// TIA Portal V17 export
// export: Created 2024-09-02T12:50:05.4870393Z, ExportSetting WithDefaults, DisplayName Totally Integrated Automation Portal, DisplayVersion V17, DisplayName TIA Portal Openness, DisplayVersion V17, DisplayName TIA Portal Version Control Interface, DisplayVersion V17, DisplayName STEP 7 Professional, DisplayVersion V17, DisplayName STEP 7 Safety, DisplayVersion V17, DisplayName WinCC Professional, DisplayVersion V17
FUNCTION_BLOCK "GraFB_Hand_01_10"   // FB1170, GRAPH
TITLE = GRAPH FB
AUTHOR : VAF
FAMILY : SK
NAME : SK
VERSION : 0.1
// Hand functions / Handfunktionen
// stored: AcknowledgeErrorsRequired true, AutoNumber true, ExtensionBlockName LTLL_ManualGraphExt, GraphVersion 4.0, InitialValuesAcquisition false, IsIECCheckEnabled false, LanguageInNetworks LAD, LockOperatingMode false, PermanentILProcessingInMANMode true, SetENOAutomatically false, SkipSteps false, UDAEnableTagReadback false, WithAlarmHandling true
   // inherited from GRAPH_BASE
   VAR
      OFF_SQ_BASE : Bool;
   END_VAR
   VAR_INPUT
      OFF_SQ : Bool;
      INIT_SQ : Bool;
      ACK_EF : Bool;
      S_PREV : Bool;
      S_NEXT : Bool;
      SW_AUTO : Bool;
      SW_TAP : Bool;
      SW_MAN : Bool;
      S_SEL : Int;
      S_ON : Bool;
      S_OFF : Bool;
      T_PUSH : Bool;
   END_VAR
   VAR_OUTPUT
      S_NO : Int;
      S_MORE : Bool;
      S_ACTIVE : Bool;
      ERR_FLT : Bool;
      AUTO_ON : Bool;
      TAP_ON : Bool;
      MAN_ON : Bool;
   END_VAR
   VAR
      extBlock { S7_SetPoint := 'True'} : "LTLL_ManualGraphExt";
   END_VAR
   VAR_TEMP
      t_FrgHand : Bool;   // Freigabe Handbetrieb / Enable manual operation
      t_Service : Bool;   // Servicebetrieb aktiv / Service operation active
   END_VAR
BEGIN
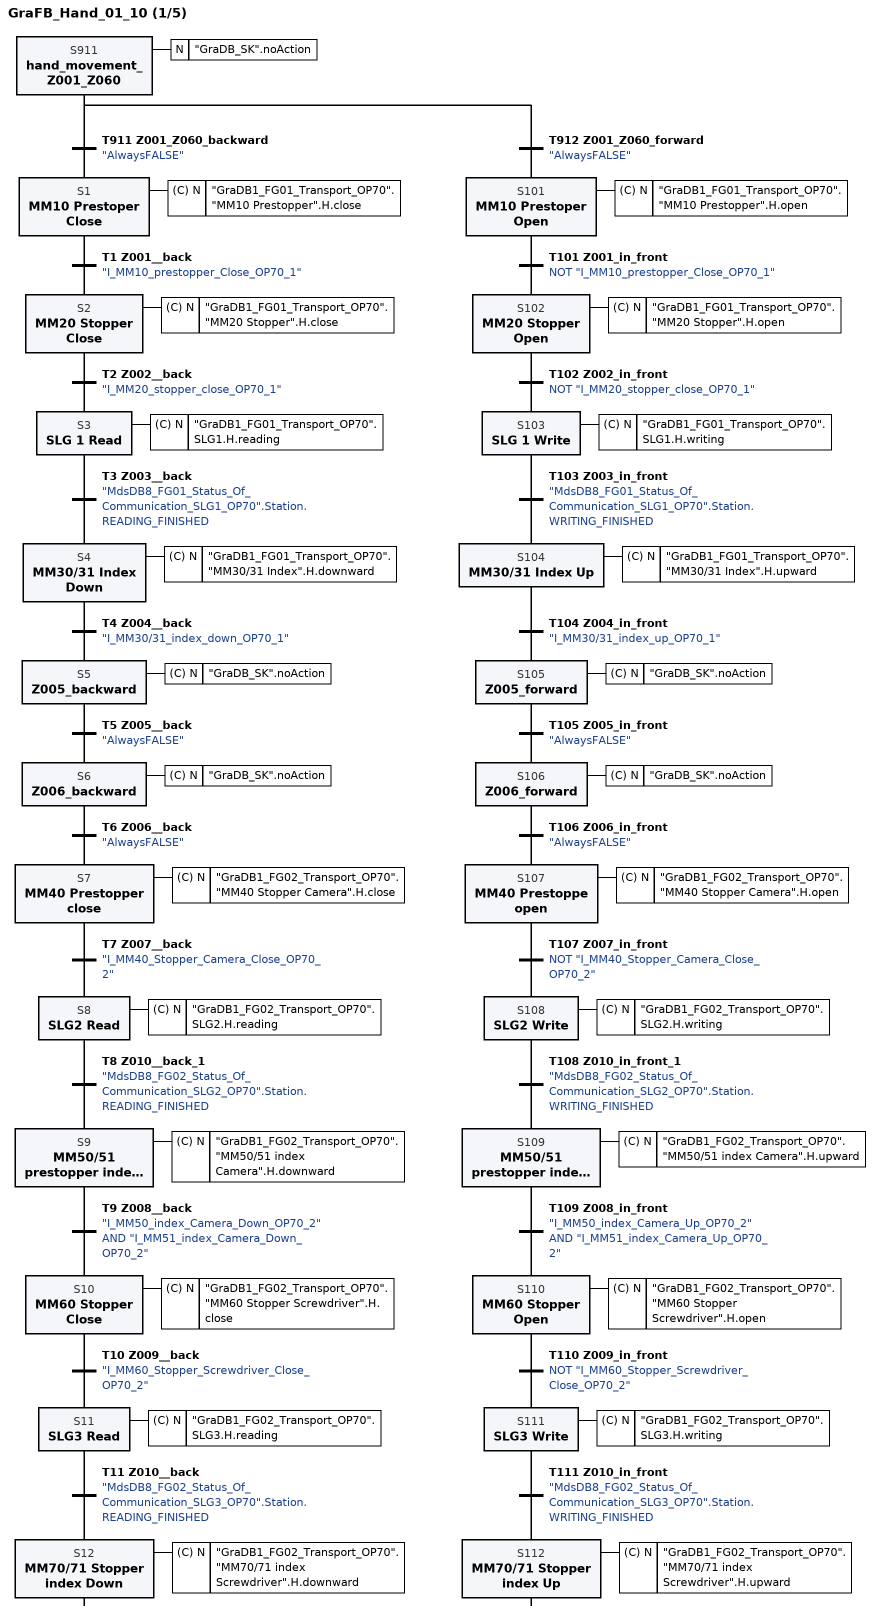
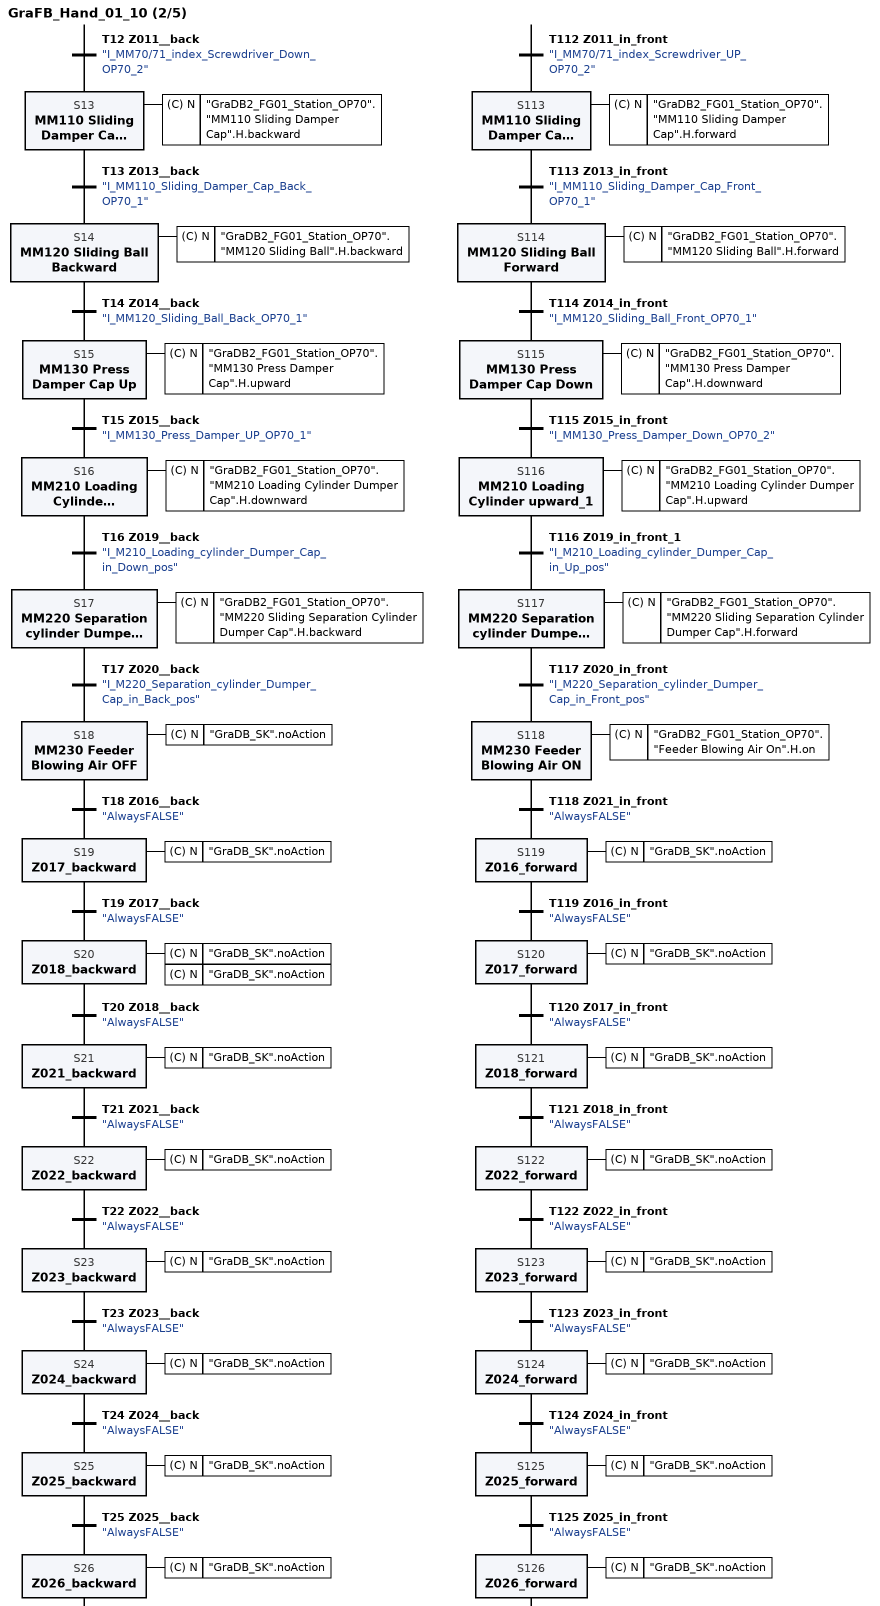
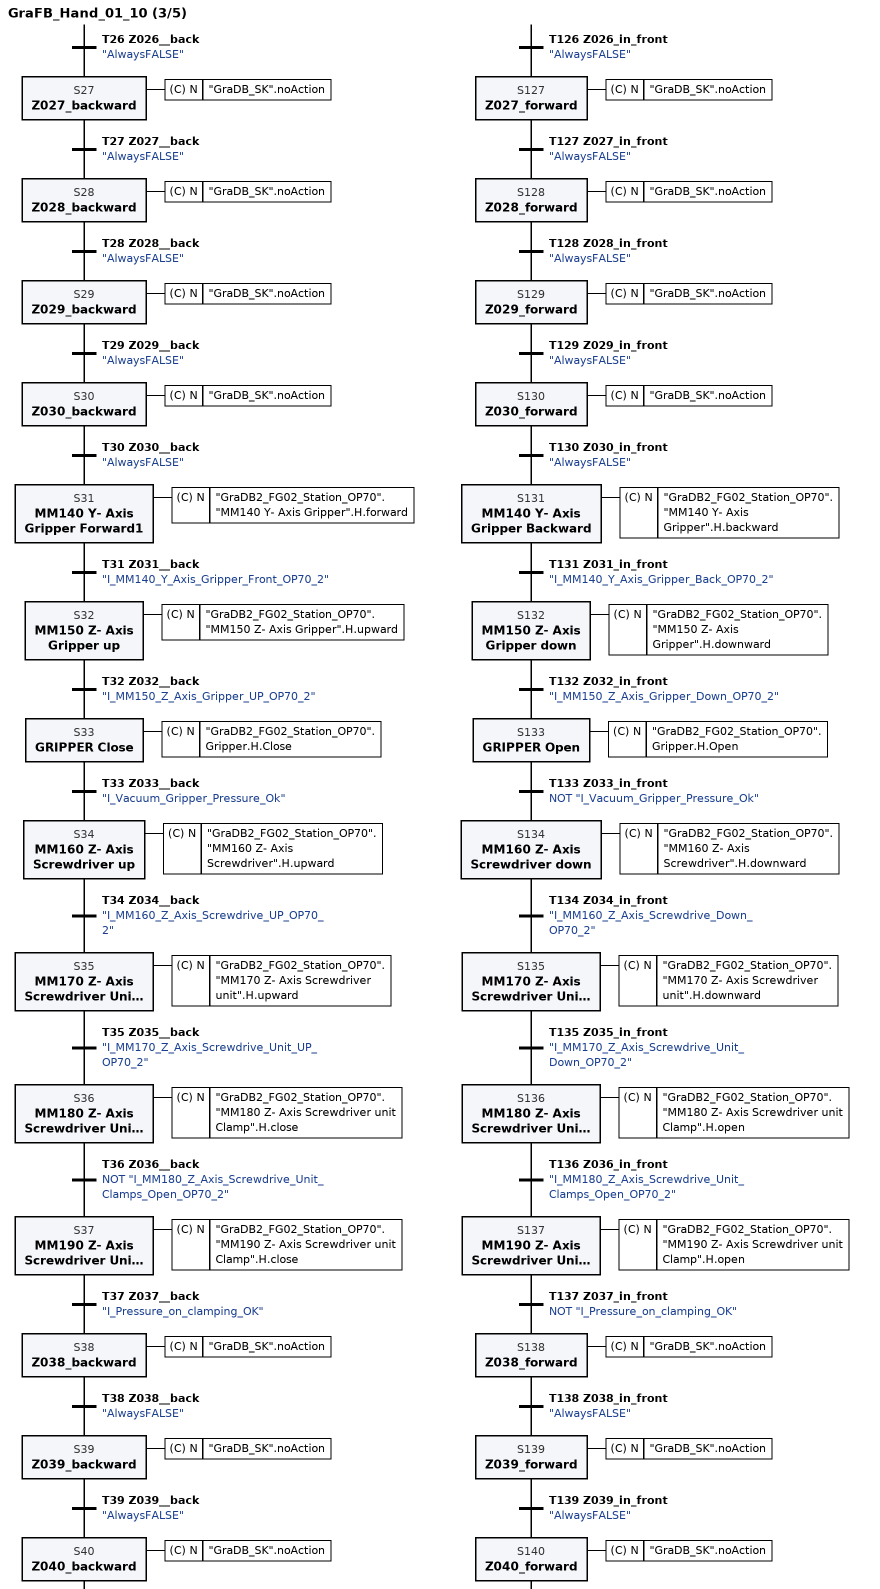
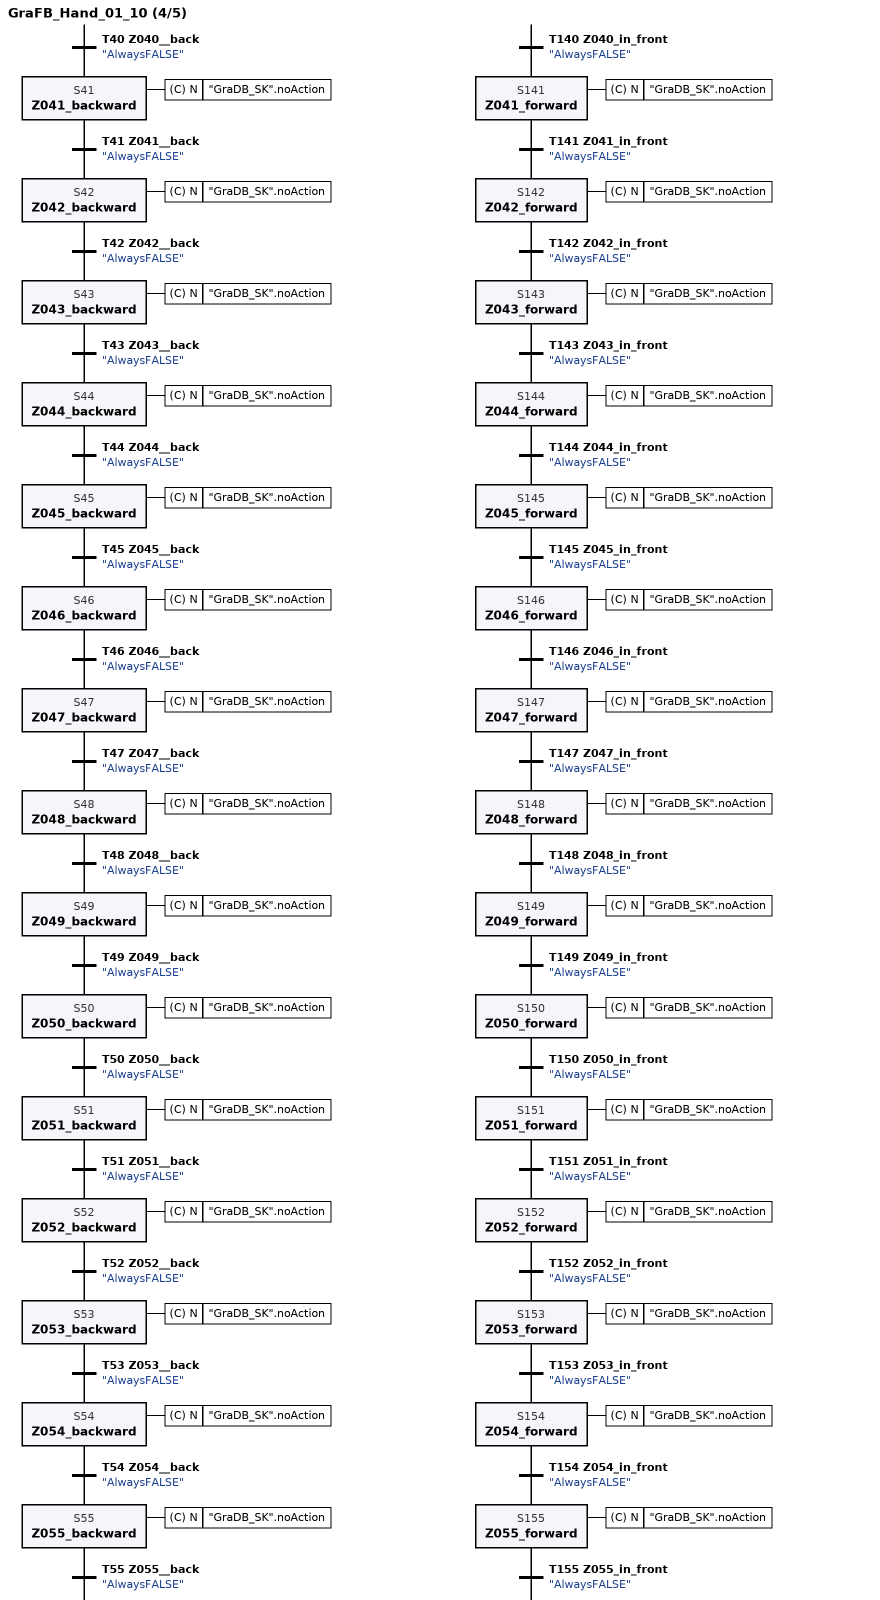
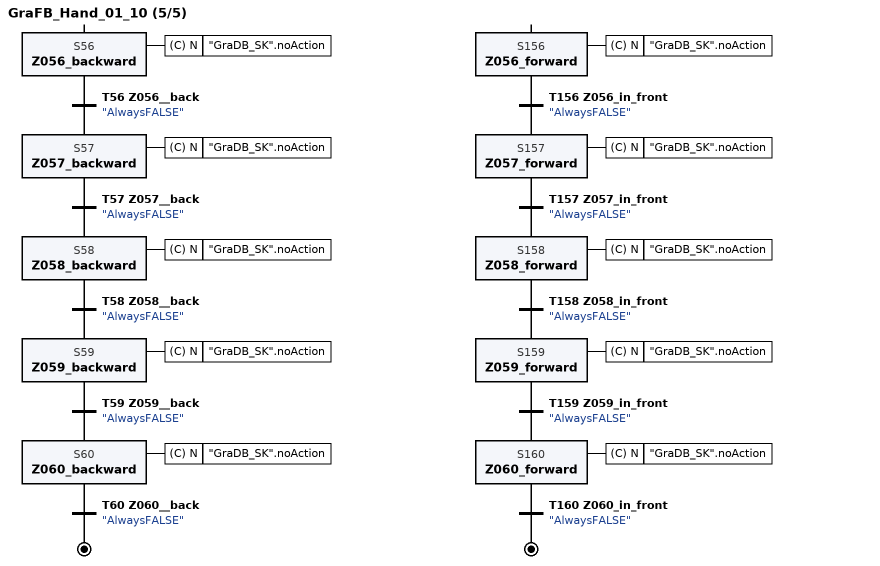
   // permanent pre-instructions
   NETWORK 1
   TITLE = HMI Lite Pass on data / HMI Lite Daten weiterreichen
      #extBlock.input := "LTLL_ManualGraphControl_OP70".screen[0].input;
   NETWORK 2
   TITLE = Instance DB Name query and pass on / Instanz DB Name abfragen und weiterreichen
      GetInstanceName(size := 0, OUT => #extBlock.input.instanceName);
   NETWORK 3
   TITLE = Interlocks Permanent machining, manual Approve and service / Interlocks Permanent Bearbeiten, Handfreigabe und Service
      IF NOT #RT_DATA.MOP.IL_PERM THEN #RT_DATA.MOP.IL_PERM := TRUE; END_IF;
      #t_FrgHand := "AnwDB_OperatingModes_OP70".BA[0]."mode_hand+start" AND "AnwDB_EKS_Data_OP70".EKS1.LEVEL_5_BK;
      #t_Service := "AnwDB_OperatingModes_OP70".BA[0].mode_service;

   // sequencer 1: Sequencer 1
   STEP hand_movement_Z001_Z060:   // S911, max time T#10S, warning time T#7S: Step commentary / Schrittkommentar
      interlock C := (none);   // hand_bereich_Z001_Z005
      supervision V := (none);   // hand_bereich_Z001_Z005
              N    "GraDB_SK".noAction
   END_STEP
   TRANSITION Z001_Z060_backward FROM hand_movement_Z001_Z060 TO "MM10 Prestoper Close"   // T911
      := "AlwaysFALSE";
   END_TRANSITION
   TRANSITION Z001_Z060_forward FROM hand_movement_Z001_Z060 TO "MM10 Prestoper Open"   // T912
      := "AlwaysFALSE";
   END_TRANSITION
   STEP "MM10 Prestoper Close":   // S1, max time T#10S, warning time T#7S
      interlock C := #t_FrgHand AND ("AlwaysTRUE" OR #t_Service);   // Z001_zur
      supervision V := NOT #Z001__back.TT AND (#"MM10 Prestoper Close".T > T#10S);   // Z001_zur
      (C)     N    "GraDB1_FG01_Transport_OP70"."MM10 Prestopper".H.close
   END_STEP
   TRANSITION Z001__back FROM "MM10 Prestoper Close" TO "MM20 Stopper Close"   // T1
      := "I_MM10_prestopper_Close_OP70_1";
   END_TRANSITION
   STEP "MM20 Stopper Close":   // S2, max time T#10S, warning time T#7S
      interlock C := #t_FrgHand AND ("AlwaysTRUE" OR #t_Service);   // Z002_zur
      supervision V := NOT #Z002__back.TT AND (#"MM20 Stopper Close".T > T#10S);   // Z002_zur
      (C)     N    "GraDB1_FG01_Transport_OP70"."MM20 Stopper".H.close
   END_STEP
   TRANSITION Z002__back FROM "MM20 Stopper Close" TO "SLG 1 Read"   // T2
      := "I_MM20_stopper_close_OP70_1";
   END_TRANSITION
   STEP "SLG 1 Read":   // S3, max time T#10S, warning time T#7S
      interlock C := #t_FrgHand AND "MdsDB8_FG01_Status_Of_Communication_SLG1_OP70".ASM.MDS_PRESENT;   // Z003_zur
      supervision V := NOT #Z003__back.TT AND (#"SLG 1 Read".T > T#10S);   // Z003_zur
      (C)     N    "GraDB1_FG01_Transport_OP70".SLG1.H.reading
   END_STEP
   TRANSITION Z003__back FROM "SLG 1 Read" TO "MM30/31 Index Down"   // T3
      := "MdsDB8_FG01_Status_Of_Communication_SLG1_OP70".Station.READING_FINISHED;
   END_TRANSITION
   STEP "MM30/31 Index Down":   // S4, max time T#10S, warning time T#7S
      interlock C := #t_FrgHand AND ("I_MM130_Press_Damper_UP_OP70_1" OR #t_Service);   // Z004_zur
      supervision V := NOT #Z004__back.TT AND (#"MM30/31 Index Down".T > T#10S);   // Z004_zur
      (C)     N    "GraDB1_FG01_Transport_OP70"."MM30/31 Index".H.downward
   END_STEP
   TRANSITION Z004__back FROM "MM30/31 Index Down" TO Z005_backward   // T4
      := "I_MM30/31_index_down_OP70_1";
   END_TRANSITION
   STEP Z005_backward:   // S5, max time T#10S, warning time T#7S
      interlock C := #t_FrgHand AND ("AlwaysFALSE" OR #t_Service);   // Z005_zur
      supervision V := NOT #Z005__back.TT AND (#Z005_backward.T > T#10S);   // Z005_zur
      (C)     N    "GraDB_SK".noAction
   END_STEP
   TRANSITION Z005__back FROM Z005_backward TO Z006_backward   // T5
      := "AlwaysFALSE";
   END_TRANSITION
   STEP "MM10 Prestoper Open":   // S101, max time T#10S, warning time T#7S
      interlock C := #t_FrgHand AND ((NOT "I_MM20_pallet_at_stopper_OP70_1" AND NOT "MdsDB8_FG01_Status_Of_Communication_SLG1_OP70".ASM.MDS_PRESENT AND "I_MM30/31_index_down_OP70_1" AND "I_MM130_Press_Damper_UP_OP70_1") OR NOT "I_MM10_pallet_at_prestopper_OP70_1" OR #t_Service);   // Z001_vor
      supervision V := NOT #Z001_in_front.TT AND (#"MM10 Prestoper Open".T > T#10S);   // Z001_vor
      (C)     N    "GraDB1_FG01_Transport_OP70"."MM10 Prestopper".H.open
   END_STEP
   TRANSITION Z001_in_front FROM "MM10 Prestoper Open" TO "MM20 Stopper Open"   // T101
      := NOT "I_MM10_prestopper_Close_OP70_1";
   END_TRANSITION
   STEP "MM20 Stopper Open":   // S102, max time T#10S, warning time T#7S
      interlock C := #t_FrgHand AND (("I_MM30/31_index_down_OP70_1" AND "I_MM130_Press_Damper_UP_OP70_1" AND NOT "I_MM40_pallet_at_Stopper_Camera_OP70_2" AND NOT "MdsDB8_FG02_Status_Of_Communication_SLG2_OP70".ASM.MDS_PRESENT AND "I_MM50_index_Camera_Down_OP70_2" AND "I_MM51_index_Camera_Down_OP70_2") OR (NOT "I_MM20_pallet_at_stopper_OP70_1" AND NOT "MdsDB8_FG01_Status_Of_Communication_SLG1_OP70".ASM.MDS_PRESENT) OR #t_Service);   // Z002_vor
      supervision V := NOT #Z002_in_front.TT AND (#"MM20 Stopper Open".T > T#10S);   // Z002_vor
      (C)     N    "GraDB1_FG01_Transport_OP70"."MM20 Stopper".H.open
   END_STEP
   TRANSITION Z002_in_front FROM "MM20 Stopper Open" TO "SLG 1 Write"   // T102
      := NOT "I_MM20_stopper_close_OP70_1";
   END_TRANSITION
   STEP "SLG 1 Write":   // S103, max time T#10S, warning time T#7S
      interlock C := #t_FrgHand AND "MdsDB8_FG01_Status_Of_Communication_SLG1_OP70".ASM.MDS_PRESENT AND "MdsDB8_FG01_Status_Of_Communication_SLG1_OP70".Station.READING_FINISHED;   // Z003_vor
      supervision V := NOT #Z003_in_front.TT AND (#"SLG 1 Write".T > T#10S);   // Z003_vor
      (C)     N    "GraDB1_FG01_Transport_OP70".SLG1.H.writing
   END_STEP
   TRANSITION Z003_in_front FROM "SLG 1 Write" TO "MM30/31 Index Up"   // T103
      := "MdsDB8_FG01_Status_Of_Communication_SLG1_OP70".Station.WRITING_FINISHED;
   END_TRANSITION
   STEP "MM30/31 Index Up":   // S104, max time T#10S, warning time T#7S
      interlock C := #t_FrgHand AND ("I_MM130_Press_Damper_UP_OP70_1" OR #t_Service);   // Z004_vor
      supervision V := NOT #Z004_in_front.TT AND (#"MM30/31 Index Up".T > T#10S);   // Z004_vor
      (C)     N    "GraDB1_FG01_Transport_OP70"."MM30/31 Index".H.upward
   END_STEP
   TRANSITION Z004_in_front FROM "MM30/31 Index Up" TO Z005_forward   // T104
      := "I_MM30/31_index_up_OP70_1";
   END_TRANSITION
   STEP Z005_forward:   // S105, max time T#10S, warning time T#7S
      interlock C := #t_FrgHand AND ("AlwaysFALSE" OR #t_Service);   // Z005_vor
      supervision V := NOT #Z005_in_front.TT AND (#Z005_forward.T > T#10S);   // Z005_vor
      (C)     N    "GraDB_SK".noAction
   END_STEP
   TRANSITION Z005_in_front FROM Z005_forward TO Z006_forward   // T105
      := "AlwaysFALSE";
   END_TRANSITION
   STEP Z006_backward:   // S6, max time T#10S, warning time T#7S: Cross transport 2 / Quertransport 2
      interlock C := #t_FrgHand AND ("AlwaysFALSE" OR #t_Service);   // Z006_zur
      supervision V := NOT #Z006__back.TT AND (#Z006_backward.T > T#10S);   // Z006_zur
      (C)     N    "GraDB_SK".noAction
   END_STEP
   TRANSITION Z006__back FROM Z006_backward TO "MM40 Prestopper close"   // T6
      := "AlwaysFALSE";
   END_TRANSITION
   STEP "MM40 Prestopper close":   // S7, max time T#10S, warning time T#7S
      interlock C := #t_FrgHand AND ("AlwaysTRUE" OR #t_Service);   // Z007_zur
      supervision V := NOT #Z007__back.TT AND (#"MM40 Prestopper close".T > T#10S);   // Z007_zur
      (C)     N    "GraDB1_FG02_Transport_OP70"."MM40 Stopper Camera".H.close
   END_STEP
   TRANSITION Z007__back FROM "MM40 Prestopper close" TO "SLG2 Read"   // T7
      := "I_MM40_Stopper_Camera_Close_OP70_2";
   END_TRANSITION
   STEP "MM50/51 prestopper index down":   // S9, max time T#10S, warning time T#7S
      interlock C := #t_FrgHand AND ("AlwaysTRUE" OR #t_Service);   // Z008_zur
      supervision V := NOT #Z008__back.TT AND (#"MM50/51 prestopper index down".T > T#10S);   // Z008_zur
      (C)     N    "GraDB1_FG02_Transport_OP70"."MM50/51 index Camera".H.downward
   END_STEP
   TRANSITION Z008__back FROM "MM50/51 prestopper index down" TO "MM60 Stopper Close"   // T9
      := "I_MM50_index_Camera_Down_OP70_2" AND "I_MM51_index_Camera_Down_OP70_2";
   END_TRANSITION
   STEP "MM60 Stopper Close":   // S10, max time T#10S, warning time T#7S
      interlock C := #t_FrgHand AND ("AlwaysTRUE" OR #t_Service);   // Z009_zur
      supervision V := NOT #Z009__back.TT AND (#"MM60 Stopper Close".T > T#10S);   // Z009_zur
      (C)     N    "GraDB1_FG02_Transport_OP70"."MM60 Stopper Screwdriver".H.close
   END_STEP
   TRANSITION Z009__back FROM "MM60 Stopper Close" TO "SLG3 Read"   // T10
      := "I_MM60_Stopper_Screwdriver_Close_OP70_2";
   END_TRANSITION
   STEP "SLG3 Read":   // S11, max time T#10S, warning time T#7S
      interlock C := #t_FrgHand AND "MdsDB8_FG02_Status_Of_Communication_SLG3_OP70".ASM.MDS_PRESENT;   // Z010_zur
      supervision V := NOT #Z010__back.TT AND (#"SLG3 Read".T > T#10S);   // Z010_zur
      (C)     N    "GraDB1_FG02_Transport_OP70".SLG3.H.reading
   END_STEP
   TRANSITION Z010__back FROM "SLG3 Read" TO "MM70/71 Stopper index Down"   // T11
      := "MdsDB8_FG02_Status_Of_Communication_SLG3_OP70".Station.READING_FINISHED;
   END_TRANSITION
   STEP Z006_forward:   // S106, max time T#10S, warning time T#7S
      interlock C := #t_FrgHand AND ("AlwaysFALSE" OR #t_Service);   // Z006_vor
      supervision V := NOT #Z006_in_front.TT AND (#Z006_forward.T > T#10S);   // Z006_vor
      (C)     N    "GraDB_SK".noAction
   END_STEP
   TRANSITION Z006_in_front FROM Z006_forward TO "MM40 Prestoppe open"   // T106
      := "AlwaysFALSE";
   END_TRANSITION
   STEP "MM40 Prestoppe open":   // S107, max time T#10S, warning time T#7S
      interlock C := #t_FrgHand AND (("I_MM50_index_Camera_Down_OP70_2" AND "I_MM51_index_Camera_Down_OP70_2" AND NOT "I_MM60_pallet_at_Stopper_Screwdriver_OP70_2" AND "I_MM70/71_index_Screwdriver_Down_OP70_2" AND "I_MM150_Z_Axis_Gripper_UP_OP70_2" AND "I_MM160_Z_Axis_Screwdrive_UP_OP70_2" AND "I_MM170_Z_Axis_Screwdrive_Unit_UP_OP70_2") OR (NOT "I_MM40_pallet_at_Stopper_Camera_OP70_2" AND NOT "MdsDB8_FG02_Status_Of_Communication_SLG2_OP70".ASM.MDS_PRESENT) OR #t_Service);   // Z007_vor
      supervision V := NOT #Z007_in_front.TT AND (#"MM40 Prestoppe open".T > T#10S);   // Z007_vor
      (C)     N    "GraDB1_FG02_Transport_OP70"."MM40 Stopper Camera".H.open
   END_STEP
   TRANSITION Z007_in_front FROM "MM40 Prestoppe open" TO "SLG2 Write"   // T107
      := NOT "I_MM40_Stopper_Camera_Close_OP70_2";
   END_TRANSITION
   STEP "MM50/51 prestopper index up":   // S109, max time T#10S, warning time T#7S
      interlock C := #t_FrgHand AND ("AlwaysTRUE" OR #t_Service);   // Z008_vor
      supervision V := NOT #Z008_in_front.TT AND (#"MM50/51 prestopper index up".T > T#10S);   // Z008_vor
      (C)     N    "GraDB1_FG02_Transport_OP70"."MM50/51 index Camera".H.upward
   END_STEP
   TRANSITION Z008_in_front FROM "MM50/51 prestopper index up" TO "MM60 Stopper Open"   // T109
      := "I_MM50_index_Camera_Up_OP70_2" AND "I_MM51_index_Camera_Up_OP70_2";
   END_TRANSITION
   STEP "MM60 Stopper Open":   // S110, max time T#10S, warning time T#7S
      interlock C := #t_FrgHand AND (("I_MM70/71_index_Screwdriver_Down_OP70_2" AND "I_MM150_Z_Axis_Gripper_UP_OP70_2" AND "I_MM160_Z_Axis_Screwdrive_UP_OP70_2" AND "I_MM170_Z_Axis_Screwdrive_Unit_UP_OP70_2" AND NOT "I_Pallet_at_Outlet_Station") OR (NOT "I_MM60_pallet_at_Stopper_Screwdriver_OP70_2" AND NOT "MdsDB8_FG02_Status_Of_Communication_SLG3_OP70".ASM.MDS_PRESENT) OR #t_Service);   // Z009_vor
      supervision V := NOT #Z009_in_front.TT AND (#"MM60 Stopper Open".T > T#10S);   // Z009_vor
      (C)     N    "GraDB1_FG02_Transport_OP70"."MM60 Stopper Screwdriver".H.open
   END_STEP
   TRANSITION Z009_in_front FROM "MM60 Stopper Open" TO "SLG3 Write"   // T110
      := NOT "I_MM60_Stopper_Screwdriver_Close_OP70_2";
   END_TRANSITION
   STEP "SLG3 Write":   // S111, max time T#10S, warning time T#7S
      interlock C := #t_FrgHand AND "MdsDB8_FG02_Status_Of_Communication_SLG3_OP70".ASM.MDS_PRESENT AND "MdsDB8_FG02_Status_Of_Communication_SLG3_OP70".Station.READING_FINISHED;   // Z010_vor
      supervision V := NOT #Z010_in_front.TT AND (#"SLG3 Write".T > T#10S);   // Z010_vor
      (C)     N    "GraDB1_FG02_Transport_OP70".SLG3.H.writing
   END_STEP
   TRANSITION Z010_in_front FROM "SLG3 Write" TO "MM70/71 Stopper index Up"   // T111
      := "MdsDB8_FG02_Status_Of_Communication_SLG3_OP70".Station.WRITING_FINISHED;
   END_TRANSITION
   STEP "MM70/71 Stopper index Down":   // S12, max time T#10S, warning time T#7S
      interlock C := #t_FrgHand AND ("AlwaysTRUE" OR #t_Service);   // Z011_zur
      supervision V := NOT #Z011__back.TT AND (#"MM70/71 Stopper index Down".T > T#10S);   // Z011_zur
      (C)     N    "GraDB1_FG02_Transport_OP70"."MM70/71 index Screwdriver".H.downward
   END_STEP
   TRANSITION Z011__back FROM "MM70/71 Stopper index Down" TO "MM110 Sliding Damper Cap Backward"   // T12
      := "I_MM70/71_index_Screwdriver_Down_OP70_2";
   END_TRANSITION
   STEP "MM120 Sliding Ball Backward":   // S14, max time T#10S, warning time T#7S
      interlock C := #t_FrgHand AND ("AlwaysTRUE" OR #t_Service);   // Z013_zur
      supervision V := NOT #Z016__back.TT AND (#"MM120 Sliding Ball Backward".T > T#10s);   // Z013_zur
      (C)     N    "GraDB2_FG01_Station_OP70"."MM120 Sliding Ball".H.backward
   END_STEP
   TRANSITION Z014__back FROM "MM120 Sliding Ball Backward" TO "MM130 Press Damper Cap Up"   // T14
      := "I_MM120_Sliding_Ball_Back_OP70_1";
   END_TRANSITION
   STEP "MM110 Sliding Damper Cap Forward":   // S113, max time T#10S, warning time T#7S
      interlock C := #t_FrgHand AND ("I_MM130_Press_Damper_UP_OP70_1" OR #t_Service);   // Z013_vor
      supervision V := NOT #Z013_in_front.TT AND (#"MM110 Sliding Damper Cap Forward".T > T#10s);   // Z013_vor
      (C)     N    "GraDB2_FG01_Station_OP70"."MM110 Sliding Damper Cap".H.forward
   END_STEP
   TRANSITION Z013_in_front FROM "MM110 Sliding Damper Cap Forward" TO "MM120 Sliding Ball Forward"   // T113
      := "I_MM110_Sliding_Damper_Cap_Front_OP70_1";
   END_TRANSITION
   STEP Z028_forward:   // S128, max time T#10S, warning time T#7S
      interlock C := #t_FrgHand AND ("AlwaysFALSE" OR #t_Service);   // Z028_vor
      supervision V := NOT #Z028_in_front.TT AND (#Z028_forward.T > T#10s);   // Z028_vor
      (C)     N    "GraDB_SK".noAction
   END_STEP
   TRANSITION Z028_in_front FROM Z028_forward TO Z029_forward   // T128
      := "AlwaysFALSE";
   END_TRANSITION
   STEP "MM70/71 Stopper index Up":   // S112, max time T#10S, warning time T#7S
      interlock C := #t_FrgHand AND (("I_MM150_Z_Axis_Gripper_UP_OP70_2" AND "I_MM160_Z_Axis_Screwdrive_UP_OP70_2" AND "I_MM170_Z_Axis_Screwdrive_Unit_UP_OP70_2") OR #t_Service);   // Z011_vor
      supervision V := NOT #Z016_in_front.TT AND (#"MM70/71 Stopper index Up".T > T#10S);   // Z011_vor
      (C)     N    "GraDB1_FG02_Transport_OP70"."MM70/71 index Screwdriver".H.upward
   END_STEP
   TRANSITION Z011_in_front FROM "MM70/71 Stopper index Up" TO "MM110 Sliding Damper Cap Forward"   // T112
      := "I_MM70/71_index_Screwdriver_UP_OP70_2";
   END_TRANSITION
   STEP "MM110 Sliding Damper Cap Backward":   // S13, max time T#10S, warning time T#7S
      interlock C := #t_FrgHand AND ("I_MM130_Press_Damper_UP_OP70_1" OR #t_Service);   // Z013_zur
      supervision V := NOT #Z016__back.TT AND (#"MM110 Sliding Damper Cap Backward".T > T#10s);   // Z013_zur
      (C)     N    "GraDB2_FG01_Station_OP70"."MM110 Sliding Damper Cap".H.backward
   END_STEP
   TRANSITION Z013__back FROM "MM110 Sliding Damper Cap Backward" TO "MM120 Sliding Ball Backward"   // T13
      := "I_MM110_Sliding_Damper_Cap_Back_OP70_1";
   END_TRANSITION
   STEP "MM130 Press Damper Cap Down":   // S115, max time T#10S, warning time T#7S
      interlock C := #t_FrgHand AND ("I_MM110_Sliding_Damper_Cap_Front_OP70_1" OR #t_Service);   // Z014_vor
      supervision V := NOT #Z015_in_front.TT AND (#"MM130 Press Damper Cap Down".T > T#10s);   // Z014_vor
      (C)     N    "GraDB2_FG01_Station_OP70"."MM130 Press Damper Cap".H.downward
   END_STEP
   TRANSITION Z015_in_front FROM "MM130 Press Damper Cap Down" TO "MM210 Loading Cylinder upward_1"   // T115
      := "I_MM130_Press_Damper_Down_OP70_2";
   END_TRANSITION
   STEP "MM230 Feeder Blowing Air OFF":   // S18, max time T#10S, warning time T#7S
      interlock C := #t_FrgHand AND ("AlwaysFALSE" OR #t_Service);   // Z016_zur
      supervision V := NOT #Z016__back.TT AND (#"MM230 Feeder Blowing Air OFF".T > T#10s);   // Z016_zur
      (C)     N    "GraDB_SK".noAction
   END_STEP
   TRANSITION Z016__back FROM "MM230 Feeder Blowing Air OFF" TO Z017_backward   // T18
      := "AlwaysFALSE";
   END_TRANSITION
   STEP Z017_backward:   // S19, max time T#10S, warning time T#7S
      interlock C := #t_FrgHand AND ("AlwaysFALSE" OR #t_Service);   // Z017_zur
      supervision V := NOT #Z017__back.TT AND (#Z017_backward.T > T#10S);   // Z017_zur
      (C)     N    "GraDB_SK".noAction
   END_STEP
   TRANSITION Z017__back FROM Z017_backward TO Z018_backward   // T19
      := "AlwaysFALSE";
   END_TRANSITION
   STEP Z018_backward:   // S20, max time T#10S, warning time T#7S
      interlock C := "AlwaysFALSE";   // Z018_zur
      supervision V := NOT #Z018__back.TT AND (#Z018_backward.T > T#10S);   // Z018_zur
      (C)     N    "GraDB_SK".noAction
      (C)     N    "GraDB_SK".noAction
   END_STEP
   TRANSITION Z018__back FROM Z018_backward TO Z021_backward   // T20
      := "AlwaysFALSE";
   END_TRANSITION
   STEP Z016_forward:   // S119, max time T#10S, warning time T#7S
      interlock C := #t_FrgHand AND ("AlwaysFALSE" OR #t_Service);   // Z016_vor
      supervision V := NOT #Z016_in_front.TT AND (#Z016_forward.T > T#10s);   // Z016_vor
      (C)     N    "GraDB_SK".noAction
   END_STEP
   TRANSITION Z016_in_front FROM Z016_forward TO Z017_forward   // T119
      := "AlwaysFALSE";
   END_TRANSITION
   STEP Z017_forward:   // S120, max time T#10S, warning time T#7S
      interlock C := #t_FrgHand AND ("AlwaysFALSE" OR #t_Service);   // Z017_vor
      supervision V := NOT #Z017_in_front.TT AND (#Z017_forward.T > T#10S);   // Z017_vor
      (C)     N    "GraDB_SK".noAction
   END_STEP
   TRANSITION Z017_in_front FROM Z017_forward TO Z018_forward   // T120
      := "AlwaysFALSE";
   END_TRANSITION
   STEP Z018_forward:   // S121, max time T#10S, warning time T#7S: "DB_F_ANW".SG_03 / "DB_F_ANW".SG_02
      interlock C := "AlwaysFALSE";   // Z018_vor
      supervision V := NOT #Z018_in_front.TT AND (#Z018_forward.T > T#10S);   // Z018_vor
      (C)     N    "GraDB_SK".noAction
   END_STEP
   TRANSITION Z018_in_front FROM Z018_forward TO Z022_forward   // T121
      := "AlwaysFALSE";
   END_TRANSITION
   STEP Z021_backward:   // S21, max time T#10S, warning time T#7S
      interlock C := #t_FrgHand AND ("AlwaysFALSE" OR #t_Service);   // Z021_zur
      supervision V := NOT #Z021__back.TT AND (#Z021_backward.T > T#10s);   // Z021_zur
      (C)     N    "GraDB_SK".noAction
   END_STEP
   TRANSITION Z021__back FROM Z021_backward TO Z022_backward   // T21
      := "AlwaysFALSE";
   END_TRANSITION
   STEP Z022_backward:   // S22, max time T#10S, warning time T#7S
      interlock C := #t_FrgHand AND ("AlwaysFALSE" OR #t_Service);   // Z022_zur
      supervision V := NOT #Z022__back.TT AND (#Z022_backward.T > T#10s);   // Z022_zur
      (C)     N    "GraDB_SK".noAction
   END_STEP
   TRANSITION Z022__back FROM Z022_backward TO Z023_backward   // T22
      := "AlwaysFALSE";
   END_TRANSITION
   STEP Z023_backward:   // S23, max time T#10S, warning time T#7S
      interlock C := #t_FrgHand AND ("AlwaysFALSE" OR #t_Service);   // Z023_zur
      supervision V := NOT #Z023__back.TT AND (#Z023_backward.T > T#10s);   // Z023_zur
      (C)     N    "GraDB_SK".noAction
   END_STEP
   TRANSITION Z023__back FROM Z023_backward TO Z024_backward   // T23
      := "AlwaysFALSE";
   END_TRANSITION
   STEP Z024_backward:   // S24, max time T#10S, warning time T#7S
      interlock C := #t_FrgHand AND ("AlwaysFALSE" OR #t_Service);   // Z024_zur
      supervision V := NOT #Z024__back.TT AND (#Z024_backward.T > T#10s);   // Z024_zur
      (C)     N    "GraDB_SK".noAction
   END_STEP
   TRANSITION Z024__back FROM Z024_backward TO Z025_backward   // T24
      := "AlwaysFALSE";
   END_TRANSITION
   STEP "MM120 Sliding Ball Forward":   // S114, max time T#10S, warning time T#7S
      interlock C := #t_FrgHand AND ("AlwaysTRUE" OR #t_Service);   // Z013_vor
      supervision V := NOT #Z014_in_front.TT AND (#"MM120 Sliding Ball Forward".T > T#10s);   // Z013_vor
      (C)     N    "GraDB2_FG01_Station_OP70"."MM120 Sliding Ball".H.forward
   END_STEP
   TRANSITION Z014_in_front FROM "MM120 Sliding Ball Forward" TO "MM130 Press Damper Cap Down"   // T114
      := "I_MM120_Sliding_Ball_Front_OP70_1";
   END_TRANSITION
   STEP Z022_forward:   // S122, max time T#10S, warning time T#7S
      interlock C := #t_FrgHand AND ("AlwaysFALSE" OR #t_Service);   // Z022_vor
      supervision V := NOT #Z022_in_front.TT AND (#Z022_forward.T > T#10s);   // Z022_vor
      (C)     N    "GraDB_SK".noAction
   END_STEP
   TRANSITION Z022_in_front FROM Z022_forward TO Z023_forward   // T122
      := "AlwaysFALSE";
   END_TRANSITION
   STEP Z023_forward:   // S123, max time T#10S, warning time T#7S
      interlock C := #t_FrgHand AND ("AlwaysFALSE" OR #t_Service);   // Z023_vor
      supervision V := NOT #Z023_in_front.TT AND (#Z023_forward.T > T#10s);   // Z023_vor
      (C)     N    "GraDB_SK".noAction
   END_STEP
   TRANSITION Z023_in_front FROM Z023_forward TO Z024_forward   // T123
      := "AlwaysFALSE";
   END_TRANSITION
   STEP Z024_forward:   // S124, max time T#10S, warning time T#7S
      interlock C := #t_FrgHand AND ("AlwaysFALSE" OR #t_Service);   // Z024_vor
      supervision V := NOT #Z024_in_front.TT AND (#Z024_forward.T > T#10s);   // Z024_vor
      (C)     N    "GraDB_SK".noAction
   END_STEP
   TRANSITION Z024_in_front FROM Z024_forward TO Z025_forward   // T124
      := "AlwaysFALSE";
   END_TRANSITION
   STEP Z025_backward:   // S25, max time T#10S, warning time T#7S
      interlock C := #t_FrgHand AND ("AlwaysFALSE" OR #t_Service);   // Z025_zur
      supervision V := NOT #Z025__back.TT AND (#Z025_backward.T > T#10s);   // Z025_zur
      (C)     N    "GraDB_SK".noAction
   END_STEP
   TRANSITION Z025__back FROM Z025_backward TO Z026_backward   // T25
      := "AlwaysFALSE";
   END_TRANSITION
   STEP Z026_backward:   // S26, max time T#10S, warning time T#7S
      interlock C := #t_FrgHand AND ("AlwaysFALSE" OR #t_Service);   // Z026_zur
      supervision V := NOT #Z026__back.TT AND (#Z026_backward.T > T#10s);   // Z026_zur
      (C)     N    "GraDB_SK".noAction
   END_STEP
   TRANSITION Z026__back FROM Z026_backward TO Z027_backward   // T26
      := "AlwaysFALSE";
   END_TRANSITION
   STEP Z027_backward:   // S27, max time T#10S, warning time T#7S
      interlock C := #t_FrgHand AND ("AlwaysFALSE" OR #t_Service);   // Z027_zur
      supervision V := NOT #Z027__back.TT AND (#Z027_backward.T > T#10s);   // Z027_zur
      (C)     N    "GraDB_SK".noAction
   END_STEP
   TRANSITION Z027__back FROM Z027_backward TO Z028_backward   // T27
      := "AlwaysFALSE";
   END_TRANSITION
   STEP "MM190 Z- Axis Screwdriver Unit Clamps Close":   // S37, max time T#10S, warning time T#7S: Step commentary / Schrittkommentar
      interlock C := "AlwaysFALSE";   // Z037_zur
      supervision V := NOT #Z037__back.TT AND (#"MM190 Z- Axis Screwdriver Unit Clamps Close".T > T#10S);   // Z037_zur
      (C)     N    "GraDB2_FG02_Station_OP70"."MM190 Z- Axis Screwdriver unit Clamp".H.close
   END_STEP
   TRANSITION Z037__back FROM "MM190 Z- Axis Screwdriver Unit Clamps Close" TO Z038_backward   // T37
      := "I_Pressure_on_clamping_OK";
   END_TRANSITION
   STEP Z029_backward:   // S29, max time T#10S, warning time T#7S
      interlock C := "AlwaysFALSE";   // Z029_zur
      supervision V := NOT #Z029__back.TT AND (#Z029_backward.T > T#10S);   // Z029_zur
      (C)     N    "GraDB_SK".noAction
   END_STEP
   TRANSITION Z029__back FROM Z029_backward TO Z030_backward   // T29
      := "AlwaysFALSE";
   END_TRANSITION
   STEP Z030_backward:   // S30, max time T#10S, warning time T#7S
      interlock C := "AlwaysFALSE";   // Z030_zur
      supervision V := NOT #Z030__back.TT AND (#Z030_backward.T > T#10S);   // Z030_zur
      (C)     N    "GraDB_SK".noAction
   END_STEP
   TRANSITION Z030__back FROM Z030_backward TO "MM140 Y- Axis Gripper Forward1"   // T30
      := "AlwaysFALSE";
   END_TRANSITION
   STEP Z026_forward:   // S126, max time T#10S, warning time T#7S
      interlock C := #t_FrgHand AND ("AlwaysFALSE" OR #t_Service);   // Z026_vor
      supervision V := NOT #Z026_in_front.TT AND (#Z026_forward.T > T#10s);   // Z026_vor
      (C)     N    "GraDB_SK".noAction
   END_STEP
   TRANSITION Z026_in_front FROM Z026_forward TO Z027_forward   // T126
      := "AlwaysFALSE";
   END_TRANSITION
   STEP Z027_forward:   // S127, max time T#10S, warning time T#7S
      interlock C := #t_FrgHand AND ("AlwaysFALSE" OR #t_Service);   // Z027_vor
      supervision V := NOT #Z027_in_front.TT AND (#Z027_forward.T > T#10s);   // Z027_vor
      (C)     N    "GraDB_SK".noAction
   END_STEP
   TRANSITION Z027_in_front FROM Z027_forward TO Z028_forward   // T127
      := "AlwaysFALSE";
   END_TRANSITION
   STEP Z028_backward:   // S28, max time T#10S, warning time T#7S
      interlock C := #t_FrgHand AND ("AlwaysTRUE" OR #t_Service);   // Z028_zur
      supervision V := NOT #Z028__back.TT AND (#Z028_backward.T > T#10s);   // Z028_zur
      (C)     N    "GraDB_SK".noAction
   END_STEP
   TRANSITION Z028__back FROM Z028_backward TO Z029_backward   // T28
      := "AlwaysFALSE";
   END_TRANSITION
   STEP Z029_forward:   // S129, max time T#10S, warning time T#7S
      interlock C := "AlwaysFALSE";   // Z029_vor
      supervision V := NOT #Z029_in_front.TT AND (#Z029_forward.T > T#10S);   // Z029_vor
      (C)     N    "GraDB_SK".noAction
   END_STEP
   TRANSITION Z029_in_front FROM Z029_forward TO Z030_forward   // T129
      := "AlwaysFALSE";
   END_TRANSITION
   STEP Z030_forward:   // S130, max time T#10S, warning time T#7S
      interlock C := "AlwaysFALSE";   // Z030_vor
      supervision V := NOT #Z030_in_front.TT AND (#Z030_forward.T > T#10S);   // Z030_vor
      (C)     N    "GraDB_SK".noAction
   END_STEP
   TRANSITION Z030_in_front FROM Z030_forward TO "MM140 Y- Axis Gripper Backward"   // T130
      := "AlwaysFALSE";
   END_TRANSITION
   STEP "MM140 Y- Axis Gripper Forward1":   // S31, max time T#10S, warning time T#7S: Step commentary / Schrittkommentar
      interlock C := #t_FrgHand AND (("I_MM150_Z_Axis_Gripper_UP_OP70_2" AND "I_MM160_Z_Axis_Screwdrive_UP_OP70_2" AND "I_MM170_Z_Axis_Screwdrive_Unit_UP_OP70_2") OR #t_Service);   // Z031_zur
      supervision V := NOT #Z031__back.TT AND (#"MM140 Y- Axis Gripper Forward1".T > T#10S);   // Z031_zur
      (C)     N    "GraDB2_FG02_Station_OP70"."MM140 Y- Axis Gripper".H.forward
   END_STEP
   TRANSITION Z031__back FROM "MM140 Y- Axis Gripper Forward1" TO "MM150 Z- Axis Gripper up"   // T31
      := "I_MM140_Y_Axis_Gripper_Front_OP70_2";
   END_TRANSITION
   STEP "MM150 Z- Axis Gripper up":   // S32, max time T#10S, warning time T#7S: Step commentary / Schrittkommentar
      interlock C := #t_FrgHand AND (("I_MM140_Y_Axis_Gripper_Back_OP70_2" AND "I_MM160_Z_Axis_Screwdrive_UP_OP70_2" AND "I_MM170_Z_Axis_Screwdrive_Unit_UP_OP70_2" AND (NOT "AnwDB_ProcessData_FG02_OP70".BEA[3].Complete.OK OR ("AnwDB_ProcessData_FG02_OP70".BEA[3].Complete.OK AND NOT "I_Vacuum_Gripper_Pressure_Ok"))) OR "I_MM140_Y_Axis_Gripper_Front_OP70_2" OR #t_Service);   // Z032_zur
      supervision V := NOT #Z032__back.TT AND (#"MM150 Z- Axis Gripper up".T > T#10S);   // Z032_zur
      (C)     N    "GraDB2_FG02_Station_OP70"."MM150 Z- Axis Gripper".H.upward
   END_STEP
   TRANSITION Z032__back FROM "MM150 Z- Axis Gripper up" TO "GRIPPER Close"   // T32
      := "I_MM150_Z_Axis_Gripper_UP_OP70_2";
   END_TRANSITION
   STEP "GRIPPER Close":   // S33, max time T#10S, warning time T#7S: Step commentary / Schrittkommentar
      interlock C := #t_FrgHand AND (NOT "AnwDB_ProcessData_FG02_OP70".BEA[3].Complete.OK OR #t_Service);   // Z033_zur
      supervision V := NOT #Z033__back.TT AND (#"GRIPPER Close".T > T#10S);   // Z033_zur
      (C)     N    "GraDB2_FG02_Station_OP70".Gripper.H.Close
   END_STEP
   TRANSITION Z033__back FROM "GRIPPER Close" TO "MM160 Z- Axis Screwdriver up"   // T33
      := "I_Vacuum_Gripper_Pressure_Ok";
   END_TRANSITION
   STEP "MM160 Z- Axis Screwdriver up":   // S34, max time T#10S, warning time T#7S: Step commentary / Schrittkommentar
      interlock C := #t_FrgHand AND ("AlwaysTRUE" OR #t_Service);   // Z034_zur
      supervision V := NOT #Z034__back.TT AND (#"MM160 Z- Axis Screwdriver up".T > T#10S);   // Z034_zur
      (C)     N    "GraDB2_FG02_Station_OP70"."MM160 Z- Axis Screwdriver".H.upward
   END_STEP
   TRANSITION Z034__back FROM "MM160 Z- Axis Screwdriver up" TO "MM170 Z- Axis Screwdriver Unit up"   // T34
      := "I_MM160_Z_Axis_Screwdrive_UP_OP70_2";
   END_TRANSITION
   STEP "MM170 Z- Axis Screwdriver Unit up":   // S35, max time T#10S, warning time T#7S: Step commentary / Schrittkommentar
      interlock C := #t_FrgHand AND ("AlwaysTRUE" OR #t_Service) AND "I_Safety_bolt_Z_Axis_Screwdrive";   // Z035_zur
      supervision V := NOT #Z035__back.TT AND (#"MM170 Z- Axis Screwdriver Unit up".T > T#10S);   // Z035_zur
      (C)     N    "GraDB2_FG02_Station_OP70"."MM170 Z- Axis Screwdriver unit".H.upward
   END_STEP
   TRANSITION Z035__back FROM "MM170 Z- Axis Screwdriver Unit up" TO "MM180 Z- Axis Screwdriver Unit Clamps Close"   // T35
      := "I_MM170_Z_Axis_Screwdrive_Unit_UP_OP70_2";
   END_TRANSITION
   STEP "MM140 Y- Axis Gripper Backward":   // S131, max time T#10S, warning time T#7S: Step commentary / Schrittkommentar
      interlock C := #t_FrgHand AND (("I_MM150_Z_Axis_Gripper_UP_OP70_2" AND "I_MM160_Z_Axis_Screwdrive_UP_OP70_2" AND "I_MM170_Z_Axis_Screwdrive_Unit_UP_OP70_2") OR #t_Service);   // Z031_vor
      supervision V := NOT #Z031_in_front.TT AND (#"MM140 Y- Axis Gripper Backward".T > T#10S);   // Z031_vor
      (C)     N    "GraDB2_FG02_Station_OP70"."MM140 Y- Axis Gripper".H.backward
   END_STEP
   TRANSITION Z031_in_front FROM "MM140 Y- Axis Gripper Backward" TO "MM150 Z- Axis Gripper down"   // T131
      := "I_MM140_Y_Axis_Gripper_Back_OP70_2";
   END_TRANSITION
   STEP "MM150 Z- Axis Gripper down":   // S132, max time T#10S, warning time T#7S: Step commentary / Schrittkommentar
      interlock C := #t_FrgHand AND ("I_MM140_Y_Axis_Gripper_Back_OP70_2" OR "I_MM140_Y_Axis_Gripper_Front_OP70_2" OR #t_Service);   // Z032_vor
      supervision V := NOT #Z032_in_front.TT AND (#"MM150 Z- Axis Gripper down".T > T#10S);   // Z032_vor
      (C)     N    "GraDB2_FG02_Station_OP70"."MM150 Z- Axis Gripper".H.downward
   END_STEP
   TRANSITION Z032_in_front FROM "MM150 Z- Axis Gripper down" TO "GRIPPER Open"   // T132
      := "I_MM150_Z_Axis_Gripper_Down_OP70_2";
   END_TRANSITION
   STEP "GRIPPER Open":   // S133, max time T#10S, warning time T#7S: Step commentary / Schrittkommentar
      interlock C := #t_FrgHand AND ((("I_MM140_Y_Axis_Gripper_Front_OP70_2" OR "I_MM140_Y_Axis_Gripper_Back_OP70_2") AND "I_MM150_Z_Axis_Gripper_Down_OP70_2" AND "I_MM70/71_index_Screwdriver_UP_OP70_2") OR #t_Service);   // Z033_vor
      supervision V := NOT #Z033_in_front.TT AND (#"GRIPPER Open".T > T#10S);   // Z033_vor
      (C)     N    "GraDB2_FG02_Station_OP70".Gripper.H.Open
   END_STEP
   TRANSITION Z033_in_front FROM "GRIPPER Open" TO "MM160 Z- Axis Screwdriver down"   // T133
      := NOT "I_Vacuum_Gripper_Pressure_Ok";
   END_TRANSITION
   STEP "MM160 Z- Axis Screwdriver down":   // S134, max time T#10S, warning time T#7S: Step commentary / Schrittkommentar
      interlock C := #t_FrgHand AND (("I_MM140_Y_Axis_Gripper_Back_OP70_2" AND "I_MM150_Z_Axis_Gripper_Down_OP70_2") OR "I_MM140_Y_Axis_Gripper_Front_OP70_2" OR #t_Service);   // Z034_vor
      supervision V := NOT #Z034_in_front.TT AND (#"MM160 Z- Axis Screwdriver down".T > T#10S);   // Z034_vor
      (C)     N    "GraDB2_FG02_Station_OP70"."MM160 Z- Axis Screwdriver".H.downward
   END_STEP
   TRANSITION Z034_in_front FROM "MM160 Z- Axis Screwdriver down" TO "MM170 Z- Axis Screwdriver Unit down"   // T134
      := "I_MM160_Z_Axis_Screwdrive_Down_OP70_2";
   END_TRANSITION
   STEP "MM170 Z- Axis Screwdriver Unit down":   // S135, max time T#10S, warning time T#7S
      interlock C := #t_FrgHand AND (((("I_MM140_Y_Axis_Gripper_Back_OP70_2" AND "I_MM150_Z_Axis_Gripper_Down_OP70_2") OR "I_MM140_Y_Axis_Gripper_Front_OP70_2") AND "I_MM160_Z_Axis_Screwdrive_UP_OP70_2") OR #t_Service) AND "I_Safety_bolt_Z_Axis_Screwdrive";   // Z035_vor
      supervision V := NOT #Z035_in_front.TT AND (#"MM170 Z- Axis Screwdriver Unit down".T > T#10S);   // Z035_vor
      (C)     N    "GraDB2_FG02_Station_OP70"."MM170 Z- Axis Screwdriver unit".H.downward
   END_STEP
   TRANSITION Z035_in_front FROM "MM170 Z- Axis Screwdriver Unit down" TO "MM180 Z- Axis Screwdriver Unit Clamps open"   // T135
      := "I_MM170_Z_Axis_Screwdrive_Unit_Down_OP70_2";
   END_TRANSITION
   STEP "MM180 Z- Axis Screwdriver Unit Clamps Close":   // S36, max time T#10S, warning time T#7S: Step commentary / Schrittkommentar
      interlock C := #t_FrgHand AND ("AlwaysFALSE" OR #t_Service);   // Z036_zur
      supervision V := NOT #Z036__back.TT AND (#"MM180 Z- Axis Screwdriver Unit Clamps Close".T > T#10S);   // Z036_zur
      (C)     N    "GraDB2_FG02_Station_OP70"."MM180 Z- Axis Screwdriver unit Clamp".H.close
   END_STEP
   TRANSITION Z036__back FROM "MM180 Z- Axis Screwdriver Unit Clamps Close" TO "MM190 Z- Axis Screwdriver Unit Clamps Close"   // T36
      := NOT "I_MM180_Z_Axis_Screwdrive_Unit_Clamps_Open_OP70_2";
   END_TRANSITION
   STEP "MM190 Z- Axis Screwdriver Unit Clamps open":   // S137, max time T#10S, warning time T#7S: Step commentary / Schrittkommentar
      interlock C := "AlwaysFALSE";   // Z037_vor
      supervision V := NOT #Z037_in_front.TT AND (#"MM190 Z- Axis Screwdriver Unit Clamps open".T > T#10S);   // Z037_vor
      (C)     N    "GraDB2_FG02_Station_OP70"."MM190 Z- Axis Screwdriver unit Clamp".H.open
   END_STEP
   TRANSITION Z037_in_front FROM "MM190 Z- Axis Screwdriver Unit Clamps open" TO Z038_forward   // T137
      := NOT "I_Pressure_on_clamping_OK";
   END_TRANSITION
   STEP Z038_forward:   // S138, max time T#10S, warning time T#7S: Step commentary / Schrittkommentar
      interlock C := "AlwaysFALSE";   // Z038_vor
      supervision V := NOT #Z038_in_front.TT AND (#Z038_forward.T > T#10S);   // Z038_vor
      (C)     N    "GraDB_SK".noAction
   END_STEP
   TRANSITION Z038_in_front FROM Z038_forward TO Z039_forward   // T138
      := "AlwaysFALSE";
   END_TRANSITION
   STEP Z039_forward:   // S139, max time T#10S, warning time T#7S: Step commentary / Schrittkommentar
      interlock C := "AlwaysFALSE";   // Z039_vor
      supervision V := NOT #Z039_in_front.TT AND (#Z039_forward.T > T#10S);   // Z039_vor
      (C)     N    "GraDB_SK".noAction
   END_STEP
   TRANSITION Z039_in_front FROM Z039_forward TO Z040_forward   // T139
      := "AlwaysFALSE";
   END_TRANSITION
   STEP Z040_forward:   // S140, max time T#10S, warning time T#7S: Step commentary / Schrittkommentar
      interlock C := "AlwaysFALSE";   // Z040_vor
      supervision V := NOT #Z040_in_front.TT AND (#Z040_forward.T > T#10S);   // Z040_vor
      (C)     N    "GraDB_SK".noAction
   END_STEP
   TRANSITION Z040_in_front FROM Z040_forward TO Z041_forward   // T140
      := "AlwaysFALSE";
   END_TRANSITION
   STEP "MM180 Z- Axis Screwdriver Unit Clamps open":   // S136, max time T#10S, warning time T#7S: Step commentary / Schrittkommentar
      interlock C := #t_FrgHand AND ("AlwaysFALSE" OR #t_Service);   // Z036_vor
      supervision V := NOT #Z036_in_front.TT AND (#"MM180 Z- Axis Screwdriver Unit Clamps open".T > T#10S);   // Z036_vor
      (C)     N    "GraDB2_FG02_Station_OP70"."MM180 Z- Axis Screwdriver unit Clamp".H.open
   END_STEP
   TRANSITION Z036_in_front FROM "MM180 Z- Axis Screwdriver Unit Clamps open" TO "MM190 Z- Axis Screwdriver Unit Clamps open"   // T136
      := "I_MM180_Z_Axis_Screwdrive_Unit_Clamps_Open_OP70_2";
   END_TRANSITION
   STEP Z041_forward:   // S141, max time T#10S, warning time T#7S: Step commentary / Schrittkommentar
      interlock C := "AlwaysFALSE";   // Z041_vor
      supervision V := NOT #Z041_in_front.TT AND (#Z041_forward.T > T#10S);   // Z041_vor
      (C)     N    "GraDB_SK".noAction
   END_STEP
   TRANSITION Z041_in_front FROM Z041_forward TO Z042_forward   // T141
      := "AlwaysFALSE";
   END_TRANSITION
   STEP Z042_backward:   // S42, max time T#10S, warning time T#7S: Step commentary / Schrittkommentar
      interlock C := "AlwaysFALSE";   // Z042_zur
      supervision V := NOT #Z042__back.TT AND (#Z042_backward.T > T#10S);   // Z042_zur
      (C)     N    "GraDB_SK".noAction
   END_STEP
   TRANSITION Z042__back FROM Z042_backward TO Z043_backward   // T42
      := "AlwaysFALSE";
   END_TRANSITION
   STEP Z043_backward:   // S43, max time T#10S, warning time T#7S: Step commentary / Schrittkommentar
      interlock C := "AlwaysFALSE";   // Z043_zur
      supervision V := NOT #Z043__back.TT AND (#Z043_backward.T > T#10S);   // Z043_zur
      (C)     N    "GraDB_SK".noAction
   END_STEP
   TRANSITION Z043__back FROM Z043_backward TO Z044_backward   // T43
      := "AlwaysFALSE";
   END_TRANSITION
   STEP Z044_backward:   // S44, max time T#10S, warning time T#7S: Step commentary / Schrittkommentar
      interlock C := "AlwaysFALSE";   // Z044_zur
      supervision V := NOT #Z044__back.TT AND (#Z044_backward.T > T#10S);   // Z044_zur
      (C)     N    "GraDB_SK".noAction
   END_STEP
   TRANSITION Z044__back FROM Z044_backward TO Z045_backward   // T44
      := "AlwaysFALSE";
   END_TRANSITION
   STEP Z045_backward:   // S45, max time T#10S, warning time T#7S: Step commentary / Schrittkommentar
      interlock C := "AlwaysFALSE";   // Z045_zur
      supervision V := NOT #Z045__back.TT AND (#Z045_backward.T > T#10S);   // Z045_zur
      (C)     N    "GraDB_SK".noAction
   END_STEP
   TRANSITION Z045__back FROM Z045_backward TO Z046_backward   // T45
      := "AlwaysFALSE";
   END_TRANSITION
   STEP Z042_forward:   // S142, max time T#10S, warning time T#7S
      interlock C := "AlwaysFALSE";   // Z042_vor
      supervision V := NOT #Z042_in_front.TT AND (#Z042_forward.T > T#10S);   // Z042_vor
      (C)     N    "GraDB_SK".noAction
   END_STEP
   TRANSITION Z042_in_front FROM Z042_forward TO Z043_forward   // T142
      := "AlwaysFALSE";
   END_TRANSITION
   STEP Z043_forward:   // S143, max time T#10S, warning time T#7S
      interlock C := "AlwaysFALSE";   // Z043_vor
      supervision V := NOT #Z043_in_front.TT AND (#Z043_forward.T > T#10S);   // Z043_vor
      (C)     N    "GraDB_SK".noAction
   END_STEP
   TRANSITION Z043_in_front FROM Z043_forward TO Z044_forward   // T143
      := "AlwaysFALSE";
   END_TRANSITION
   STEP Z044_forward:   // S144, max time T#10S, warning time T#7S
      interlock C := "AlwaysFALSE";   // Z044_vor
      supervision V := NOT #Z044_in_front.TT AND (#Z044_forward.T > T#10S);   // Z044_vor
      (C)     N    "GraDB_SK".noAction
   END_STEP
   TRANSITION Z044_in_front FROM Z044_forward TO Z045_forward   // T144
      := "AlwaysFALSE";
   END_TRANSITION
   STEP Z045_forward:   // S145, max time T#10S, warning time T#7S
      interlock C := "AlwaysFALSE";   // Z045_vor
      supervision V := NOT #Z045_in_front.TT AND (#Z045_forward.T > T#10S);   // Z045_vor
      (C)     N    "GraDB_SK".noAction
   END_STEP
   TRANSITION Z045_in_front FROM Z045_forward TO Z046_forward   // T145
      := "AlwaysFALSE";
   END_TRANSITION
   STEP Z046_backward:   // S46, max time T#10S, warning time T#7S: Step commentary / Schrittkommentar
      interlock C := "AlwaysFALSE";   // Z046_zur
      supervision V := NOT #Z046__back.TT AND (#Z046_backward.T > T#10S);   // Z046_zur
      (C)     N    "GraDB_SK".noAction
   END_STEP
   TRANSITION Z046__back FROM Z046_backward TO Z047_backward   // T46
      := "AlwaysFALSE";
   END_TRANSITION
   STEP Z047_backward:   // S47, max time T#10S, warning time T#7S: Step commentary / Schrittkommentar
      interlock C := "AlwaysFALSE";   // Z047_zur
      supervision V := NOT #Z047__back.TT AND (#Z047_backward.T > T#10S);   // Z047_zur
      (C)     N    "GraDB_SK".noAction
   END_STEP
   TRANSITION Z047__back FROM Z047_backward TO Z048_backward   // T47
      := "AlwaysFALSE";
   END_TRANSITION
   STEP Z048_backward:   // S48, max time T#10S, warning time T#7S: Step commentary / Schrittkommentar
      interlock C := "AlwaysFALSE";   // Z048_zur
      supervision V := NOT #Z048__back.TT AND (#Z048_backward.T > T#10S);   // Z048_zur
      (C)     N    "GraDB_SK".noAction
   END_STEP
   TRANSITION Z048__back FROM Z048_backward TO Z049_backward   // T48
      := "AlwaysFALSE";
   END_TRANSITION
   STEP Z049_backward:   // S49, max time T#10S, warning time T#7S: Step commentary / Schrittkommentar
      interlock C := "AlwaysFALSE";   // Z049_zur
      supervision V := NOT #Z049__back.TT AND (#Z049_backward.T > T#10S);   // Z049_zur
      (C)     N    "GraDB_SK".noAction
   END_STEP
   TRANSITION Z049__back FROM Z049_backward TO Z050_backward   // T49
      := "AlwaysFALSE";
   END_TRANSITION
   STEP Z050_backward:   // S50, max time T#10S, warning time T#7S: Step commentary / Schrittkommentar
      interlock C := "AlwaysFALSE";   // Z050_zur
      supervision V := NOT #Z050__back.TT AND (#Z050_backward.T > T#10S);   // Z050_zur
      (C)     N    "GraDB_SK".noAction
   END_STEP
   TRANSITION Z050__back FROM Z050_backward TO Z051_backward   // T50
      := "AlwaysFALSE";
   END_TRANSITION
   STEP Z046_forward:   // S146, max time T#10S, warning time T#7S: Step commentary / Schrittkommentar
      interlock C := "AlwaysFALSE";   // Z046_vor
      supervision V := NOT #Z046_in_front.TT AND (#Z046_forward.T > T#10S);   // Z046_vor
      (C)     N    "GraDB_SK".noAction
   END_STEP
   TRANSITION Z046_in_front FROM Z046_forward TO Z047_forward   // T146
      := "AlwaysFALSE";
   END_TRANSITION
   STEP Z047_forward:   // S147, max time T#10S, warning time T#7S: Step commentary / Schrittkommentar
      interlock C := "AlwaysFALSE";   // Z047_vor
      supervision V := NOT #Z047_in_front.TT AND (#Z047_forward.T > T#10S);   // Z047_vor
      (C)     N    "GraDB_SK".noAction
   END_STEP
   TRANSITION Z047_in_front FROM Z047_forward TO Z048_forward   // T147
      := "AlwaysFALSE";
   END_TRANSITION
   STEP Z048_forward:   // S148, max time T#10S, warning time T#7S: Step commentary / Schrittkommentar
      interlock C := "AlwaysFALSE";   // Z048_vor
      supervision V := NOT #Z048_in_front.TT AND (#Z048_forward.T > T#10S);   // Z048_vor
      (C)     N    "GraDB_SK".noAction
   END_STEP
   TRANSITION Z048_in_front FROM Z048_forward TO Z049_forward   // T148
      := "AlwaysFALSE";
   END_TRANSITION
   STEP Z049_forward:   // S149, max time T#10S, warning time T#7S: Step commentary / Schrittkommentar
      interlock C := "AlwaysFALSE";   // Z049_vor
      supervision V := NOT #Z049_in_front.TT AND (#Z049_forward.T > T#10S);   // Z049_vor
      (C)     N    "GraDB_SK".noAction
   END_STEP
   TRANSITION Z049_in_front FROM Z049_forward TO Z050_forward   // T149
      := "AlwaysFALSE";
   END_TRANSITION
   STEP Z050_forward:   // S150, max time T#10S, warning time T#7S: Step commentary / Schrittkommentar
      interlock C := "AlwaysFALSE";   // Z050_vor
      supervision V := NOT #Z050_in_front.TT AND (#Z050_forward.T > T#10S);   // Z050_vor
      (C)     N    "GraDB_SK".noAction
   END_STEP
   TRANSITION Z050_in_front FROM Z050_forward TO Z051_forward   // T150
      := "AlwaysFALSE";
   END_TRANSITION
   STEP Z051_backward:   // S51, max time T#10S, warning time T#7S: Step commentary / Schrittkommentar
      interlock C := "AlwaysFALSE";   // Z051_zur
      supervision V := NOT #Z051__back.TT AND (#Z051_backward.T > T#10S);   // Z051_zur
      (C)     N    "GraDB_SK".noAction
   END_STEP
   TRANSITION Z051__back FROM Z051_backward TO Z052_backward   // T51
      := "AlwaysFALSE";
   END_TRANSITION
   STEP Z052_backward:   // S52, max time T#10S, warning time T#7S: Step commentary / Schrittkommentar
      interlock C := "AlwaysFALSE";   // Z052_zur
      supervision V := NOT #Z052__back.TT AND (#Z052_backward.T > T#10S);   // Z052_zur
      (C)     N    "GraDB_SK".noAction
   END_STEP
   TRANSITION Z052__back FROM Z052_backward TO Z053_backward   // T52
      := "AlwaysFALSE";
   END_TRANSITION
   STEP Z053_backward:   // S53, max time T#10S, warning time T#7S: Step commentary / Schrittkommentar
      interlock C := "AlwaysFALSE";   // Z053_zur
      supervision V := NOT #Z053__back.TT AND (#Z053_backward.T > T#10S);   // Z053_zur
      (C)     N    "GraDB_SK".noAction
   END_STEP
   TRANSITION Z053__back FROM Z053_backward TO Z054_backward   // T53
      := "AlwaysFALSE";
   END_TRANSITION
   STEP Z054_backward:   // S54, max time T#10S, warning time T#7S: Step commentary / Schrittkommentar
      interlock C := "AlwaysFALSE";   // Z054_zur
      supervision V := NOT #Z054__back.TT AND (#Z054_backward.T > T#10S);   // Z054_zur
      (C)     N    "GraDB_SK".noAction
   END_STEP
   TRANSITION Z054__back FROM Z054_backward TO Z055_backward   // T54
      := "AlwaysFALSE";
   END_TRANSITION
   STEP Z055_backward:   // S55, max time T#10S, warning time T#7S: Step commentary / Schrittkommentar
      interlock C := "AlwaysFALSE";   // Z055_zur
      supervision V := NOT #Z055__back.TT AND (#Z055_backward.T > T#10S);   // Z055_zur
      (C)     N    "GraDB_SK".noAction
   END_STEP
   TRANSITION Z055__back FROM Z055_backward TO Z056_backward   // T55
      := "AlwaysFALSE";
   END_TRANSITION
   STEP Z056_backward:   // S56, max time T#10S, warning time T#7S: Step commentary / Schrittkommentar
      interlock C := "AlwaysFALSE";   // Z056_zur
      supervision V := NOT #Z056__back.TT AND (#Z056_backward.T > T#10S);   // Z056_zur
      (C)     N    "GraDB_SK".noAction
   END_STEP
   TRANSITION Z056__back FROM Z056_backward TO Z057_backward   // T56
      := "AlwaysFALSE";
   END_TRANSITION
   STEP Z057_backward:   // S57, max time T#10S, warning time T#7S: Step commentary / Schrittkommentar
      interlock C := (none);   // Z057_zur
      supervision V := NOT #Z057__back.TT AND (#Z057_backward.T > T#10S);   // Z057_zur
      (C)     N    "GraDB_SK".noAction
   END_STEP
   TRANSITION Z057__back FROM Z057_backward TO Z058_backward   // T57
      := "AlwaysFALSE";
   END_TRANSITION
   STEP Z058_backward:   // S58, max time T#10S, warning time T#7S: Step commentary / Schrittkommentar
      interlock C := "AlwaysFALSE";   // Z058_zur
      supervision V := NOT #Z058__back.TT AND (#Z058_backward.T > T#10S);   // Z058_zur
      (C)     N    "GraDB_SK".noAction
   END_STEP
   TRANSITION Z058__back FROM Z058_backward TO Z059_backward   // T58
      := "AlwaysFALSE";
   END_TRANSITION
   STEP Z059_backward:   // S59, max time T#10S, warning time T#7S: Step commentary / Schrittkommentar
      interlock C := "AlwaysFALSE";   // Z059_zur
      supervision V := NOT #Z059__back.TT AND (#Z059_backward.T > T#10S);   // Z059_zur
      (C)     N    "GraDB_SK".noAction
   END_STEP
   TRANSITION Z059__back FROM Z059_backward TO Z060_backward   // T59
      := "AlwaysFALSE";
   END_TRANSITION
   STEP Z060_backward:   // S60, max time T#10S, warning time T#7S: Step commentary / Schrittkommentar
      interlock C := "AlwaysFALSE";   // Z060_zur
      supervision V := NOT #Z060__back.TT AND (#Z060_backward.T > T#10S);   // Z060_zur
      (C)     N    "GraDB_SK".noAction
   END_STEP
   TRANSITION Z060__back FROM Z060_backward TO END   // T60
      := "AlwaysFALSE";
   END_TRANSITION
   STEP Z051_forward:   // S151, max time T#10S, warning time T#7S
      interlock C := "AlwaysFALSE";   // Z051_vor
      supervision V := NOT #Z051_in_front.TT AND (#Z051_forward.T > T#10S);   // Z051_vor
      (C)     N    "GraDB_SK".noAction
   END_STEP
   TRANSITION Z051_in_front FROM Z051_forward TO Z052_forward   // T151
      := "AlwaysFALSE";
   END_TRANSITION
   STEP Z052_forward:   // S152, max time T#10S, warning time T#7S
      interlock C := "AlwaysFALSE";   // Z052_vor
      supervision V := NOT #Z052_in_front.TT AND (#Z052_forward.T > T#10S);   // Z052_vor
      (C)     N    "GraDB_SK".noAction
   END_STEP
   TRANSITION Z052_in_front FROM Z052_forward TO Z053_forward   // T152
      := "AlwaysFALSE";
   END_TRANSITION
   STEP Z053_forward:   // S153, max time T#10S, warning time T#7S
      interlock C := "AlwaysFALSE";   // Z053_vor
      supervision V := NOT #Z053_in_front.TT AND (#Z053_forward.T > T#10S);   // Z053_vor
      (C)     N    "GraDB_SK".noAction
   END_STEP
   TRANSITION Z053_in_front FROM Z053_forward TO Z054_forward   // T153
      := "AlwaysFALSE";
   END_TRANSITION
   STEP Z054_forward:   // S154, max time T#10S, warning time T#7S
      interlock C := "AlwaysFALSE";   // Z054_vor
      supervision V := NOT #Z054_in_front.TT AND (#Z054_forward.T > T#10S);   // Z054_vor
      (C)     N    "GraDB_SK".noAction
   END_STEP
   TRANSITION Z054_in_front FROM Z054_forward TO Z055_forward   // T154
      := "AlwaysFALSE";
   END_TRANSITION
   STEP Z055_forward:   // S155, max time T#10S, warning time T#7S
      interlock C := "AlwaysFALSE";   // Z055_vor
      supervision V := NOT #Z055_in_front.TT AND (#Z055_forward.T > T#10S);   // Z055_vor
      (C)     N    "GraDB_SK".noAction
   END_STEP
   TRANSITION Z055_in_front FROM Z055_forward TO Z056_forward   // T155
      := "AlwaysFALSE";
   END_TRANSITION
   STEP Z056_forward:   // S156, max time T#10S, warning time T#7S: Step commentary / Schrittkommentar
      interlock C := "AlwaysFALSE";   // Z056_vor
      supervision V := NOT #Z056_in_front.TT AND (#Z056_forward.T > T#10S);   // Z056_vor
      (C)     N    "GraDB_SK".noAction
   END_STEP
   TRANSITION Z056_in_front FROM Z056_forward TO Z057_forward   // T156
      := "AlwaysFALSE";
   END_TRANSITION
   STEP Z057_forward:   // S157, max time T#10S, warning time T#7S: Step commentary / Schrittkommentar
      interlock C := "AlwaysFALSE";   // Z057_vor
      supervision V := NOT #Z057_in_front.TT AND (#Z057_forward.T > T#10S);   // Z057_vor
      (C)     N    "GraDB_SK".noAction
   END_STEP
   TRANSITION Z057_in_front FROM Z057_forward TO Z058_forward   // T157
      := "AlwaysFALSE";
   END_TRANSITION
   STEP Z058_forward:   // S158, max time T#10S, warning time T#7S: Step commentary / Schrittkommentar
      interlock C := "AlwaysFALSE";   // Z058_vor
      supervision V := NOT #Z058_in_front.TT AND (#Z058_forward.T > T#10S);   // Z058_vor
      (C)     N    "GraDB_SK".noAction
   END_STEP
   TRANSITION Z058_in_front FROM Z058_forward TO Z059_forward   // T158
      := "AlwaysFALSE";
   END_TRANSITION
   STEP Z059_forward:   // S159, max time T#10S, warning time T#7S: Step commentary / Schrittkommentar
      interlock C := "AlwaysFALSE";   // Z059_vor
      supervision V := NOT #Z059_in_front.TT AND (#Z059_forward.T > T#10S);   // Z059_vor
      (C)     N    "GraDB_SK".noAction
   END_STEP
   TRANSITION Z059_in_front FROM Z059_forward TO Z060_forward   // T159
      := "AlwaysFALSE";
   END_TRANSITION
   STEP Z060_forward:   // S160, max time T#10S, warning time T#7S: Step commentary / Schrittkommentar
      interlock C := "AlwaysFALSE";   // Z060_vor
      supervision V := NOT #Z060_in_front.TT AND (#Z060_forward.T > T#10S);   // Z060_vor
      (C)     N    "GraDB_SK".noAction
   END_STEP
   TRANSITION Z060_in_front FROM Z060_forward TO END   // T160
      := "AlwaysFALSE";
   END_TRANSITION
   STEP Z025_forward:   // S125, max time T#10S, warning time T#7S
      interlock C := #t_FrgHand AND ("AlwaysFALSE" OR #t_Service);   // Z025_vor
      supervision V := NOT #Z025_in_front.TT AND (#Z025_forward.T > T#10s);   // Z025_vor
      (C)     N    "GraDB_SK".noAction
   END_STEP
   TRANSITION Z025_in_front FROM Z025_forward TO Z026_forward   // T125
      := "AlwaysFALSE";
   END_TRANSITION
   STEP "MM130 Press Damper Cap Up":   // S15, max time T#10S, warning time T#7S
      interlock C := #t_FrgHand AND ("AlwaysTRUE" OR #t_Service);   // Z014_zur
      supervision V := NOT #Z015__back.TT AND (#"MM130 Press Damper Cap Up".T > T#10s);   // Z014_zur
      (C)     N    "GraDB2_FG01_Station_OP70"."MM130 Press Damper Cap".H.upward
   END_STEP
   TRANSITION Z015__back FROM "MM130 Press Damper Cap Up" TO "MM210 Loading Cylinder Downward"   // T15
      := "I_MM130_Press_Damper_UP_OP70_1";
   END_TRANSITION
   STEP Z038_backward:   // S38, max time T#10S, warning time T#7S: Step commentary / Schrittkommentar
      interlock C := "AlwaysFALSE";   // Z038_zur
      supervision V := NOT #Z038__back.TT AND (#Z038_backward.T > T#10S);   // Z038_zur
      (C)     N    "GraDB_SK".noAction
   END_STEP
   TRANSITION Z038__back FROM Z038_backward TO Z039_backward   // T38
      := "AlwaysFALSE";
   END_TRANSITION
   STEP Z039_backward:   // S39, max time T#10S, warning time T#7S: Step commentary / Schrittkommentar
      interlock C := "AlwaysFALSE";   // Z039_zur
      supervision V := NOT #Z039__back.TT AND (#Z039_backward.T > T#10S);   // Z039_zur
      (C)     N    "GraDB_SK".noAction
   END_STEP
   TRANSITION Z039__back FROM Z039_backward TO Z040_backward   // T39
      := "AlwaysFALSE";
   END_TRANSITION
   STEP Z040_backward:   // S40, max time T#10S, warning time T#7S: Step commentary / Schrittkommentar
      interlock C := "AlwaysFALSE";   // Z040_zur
      supervision V := NOT #Z040__back.TT AND (#Z040_backward.T > T#10S);   // Z040_zur
      (C)     N    "GraDB_SK".noAction
   END_STEP
   TRANSITION Z040__back FROM Z040_backward TO Z041_backward   // T40
      := "AlwaysFALSE";
   END_TRANSITION
   STEP Z041_backward:   // S41, max time T#10S, warning time T#7S: Step commentary / Schrittkommentar
      interlock C := "AlwaysFALSE";   // Z041_zur
      supervision V := NOT #Z041__back.TT AND (#Z041_backward.T > T#10S);   // Z041_zur
      (C)     N    "GraDB_SK".noAction
   END_STEP
   TRANSITION Z041__back FROM Z041_backward TO Z042_backward   // T41
      := "AlwaysFALSE";
   END_TRANSITION
   STEP "SLG2 Read":   // S8, max time T#10S, warning time T#7S
      interlock C := #t_FrgHand AND "MdsDB8_FG02_Status_Of_Communication_SLG2_OP70".ASM.MDS_PRESENT;   // Z010_zur
      supervision V := NOT #Z010__back_1.TT AND (#"SLG2 Read".T > T#10S);   // Z010_zur
      (C)     N    "GraDB1_FG02_Transport_OP70".SLG2.H.reading
   END_STEP
   TRANSITION Z010__back_1 FROM "SLG2 Read" TO "MM50/51 prestopper index down"   // T8
      := "MdsDB8_FG02_Status_Of_Communication_SLG2_OP70".Station.READING_FINISHED;
   END_TRANSITION
   STEP "SLG2 Write":   // S108, max time T#10S, warning time T#7S
      interlock C := #t_FrgHand AND "MdsDB8_FG02_Status_Of_Communication_SLG2_OP70".ASM.MDS_PRESENT AND "MdsDB8_FG02_Status_Of_Communication_SLG2_OP70".Station.READING_FINISHED;   // Z010_vor
      supervision V := NOT #Z010_in_front_1.TT AND (#"SLG2 Write".T > T#10S);   // Z010_vor
      (C)     N    "GraDB1_FG02_Transport_OP70".SLG2.H.writing
   END_STEP
   TRANSITION Z010_in_front_1 FROM "SLG2 Write" TO "MM50/51 prestopper index up"   // T108
      := "MdsDB8_FG02_Status_Of_Communication_SLG2_OP70".Station.WRITING_FINISHED;
   END_TRANSITION
   STEP "MM220 Separation cylinder Dumper Cap Forward":   // S117, max time T#10S, warning time T#7S
      interlock C := #t_FrgHand AND ("AlwaysTRUE" OR #t_Service);   // Z020_vor
      supervision V := NOT #Z020_in_front.TT AND (#"MM220 Separation cylinder Dumper Cap Forward".T > T#10s);   // Z020_vor
      (C)     N    "GraDB2_FG01_Station_OP70"."MM220 Sliding Separation Cylinder Dumper Cap".H.forward
   END_STEP
   TRANSITION Z020_in_front FROM "MM220 Separation cylinder Dumper Cap Forward" TO "MM230 Feeder Blowing Air ON"   // T117
      := "I_M220_Separation_cylinder_Dumper_Cap_in_Front_pos";
   END_TRANSITION
   STEP "MM230 Feeder Blowing Air ON":   // S118, max time T#10S, warning time T#7S
      interlock C := #t_FrgHand AND (NOT "GraDB2_FG01_Station_OP70".Feeder_Damper_Cap.Status.Part_insite OR #t_Service);   // Z021_vor
      supervision V := NOT #Z021_in_front.TT AND (#"MM230 Feeder Blowing Air ON".T > T#10s);   // Z021_vor
      (C)     N    "GraDB2_FG01_Station_OP70"."Feeder Blowing Air On".H.on
   END_STEP
   TRANSITION Z021_in_front FROM "MM230 Feeder Blowing Air ON" TO Z016_forward   // T118
      := "AlwaysFALSE";
   END_TRANSITION
   STEP "MM210 Loading Cylinder Downward":   // S16, max time T#10S, warning time T#7S
      interlock C := #t_FrgHand AND ("AlwaysTRUE" OR #t_Service);   // Z019_zur
      supervision V := NOT #Z019__back.TT AND (#"MM210 Loading Cylinder Downward".T > T#10s);   // Z019_zur
      (C)     N    "GraDB2_FG01_Station_OP70"."MM210 Loading Cylinder Dumper Cap".H.downward
   END_STEP
   TRANSITION Z019__back FROM "MM210 Loading Cylinder Downward" TO "MM220 Separation cylinder Dumper Cap Backward"   // T16
      := "I_M210_Loading_cylinder_Dumper_Cap_in_Down_pos";
   END_TRANSITION
   STEP "MM220 Separation cylinder Dumper Cap Backward":   // S17, max time T#10S, warning time T#7S
      interlock C := #t_FrgHand AND ((NOT "GraDB2_FG01_Station_OP70".Feeder_Damper_Cap.Status.Part_in_Separator AND NOT "GraDB2_FG01_Station_OP70".Feeder_Damper_Cap.Status.Part_in_pipe) OR #t_Service);   // Z020_zur
      supervision V := NOT #Z020__back.TT AND (#"MM220 Separation cylinder Dumper Cap Backward".T > T#10s);   // Z020_zur
      (C)     N    "GraDB2_FG01_Station_OP70"."MM220 Sliding Separation Cylinder Dumper Cap".H.backward
   END_STEP
   TRANSITION Z020__back FROM "MM220 Separation cylinder Dumper Cap Backward" TO "MM230 Feeder Blowing Air OFF"   // T17
      := "I_M220_Separation_cylinder_Dumper_Cap_in_Back_pos";
   END_TRANSITION
   STEP "MM210 Loading Cylinder upward_1":   // S116, max time T#10S, warning time T#7S
      interlock C := #t_FrgHand AND ("AlwaysTRUE" OR #t_Service);   // Z019_vor
      supervision V := NOT #Z019_in_front_1.TT AND (#"MM210 Loading Cylinder upward_1".T > T#10s);   // Z019_vor
      (C)     N    "GraDB2_FG01_Station_OP70"."MM210 Loading Cylinder Dumper Cap".H.upward
   END_STEP
   TRANSITION Z019_in_front_1 FROM "MM210 Loading Cylinder upward_1" TO "MM220 Separation cylinder Dumper Cap Forward"   // T116
      := "I_M210_Loading_cylinder_Dumper_Cap_in_Up_pos";
   END_TRANSITION

   // permanent post-instructions
   NETWORK 1
   TITLE = HMI Lite Pass on data / HMI Lite Daten weiterreichen
      "LTLL_ManualGraphInterlock"(ManualGraphExtOutput := #extBlock.output,
                              ManualGraphControlScreen := "LTLL_ManualGraphControl_OP70".screen[0]);
   NETWORK 2
   TITLE = Report step error / Schrittkettenfehler melden
      "SysFC_NumOfSQErrors"(FLT := #RT_DATA.SQ_FLAGS.ERR_FLT,
                            Fault_SQ := "AnwDB_OperatingModes_OP70".BA[0].error_report_SK,
                            NumOf_Fault_SQ := "AnwDB_ZP_Alarm_OP70".FaultsNoSK_ST1);
END_FUNCTION_BLOCK
